FUNCTION_BLOCK P_Call (* Calls one atomic skill: latches P1..P4 on EI, continues on DONE (EO) or FAILED (ERR); ignores completions it did not request *)
  (* Standard: 61499-2 *)
  (* Version 2.0, 2026-09-27, Project contributors, Filling cell reference model *)
  PACKAGE fillingcell;
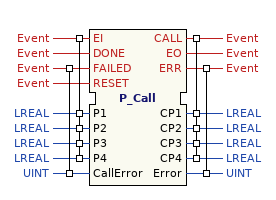
  EVENT_INPUT
    EI WITH P1, P2, P3, P4;
    DONE;
    FAILED WITH CallError;
    RESET;
  END_EVENT
  EVENT_OUTPUT
    CALL WITH CP1, CP2, CP3, CP4;
    EO;
    ERR WITH Error;
  END_EVENT
  VAR_INPUT
    P1 : LREAL;
    P2 : LREAL;
    P3 : LREAL;
    P4 : LREAL;
    CallError : UINT;
  END_VAR
  VAR_OUTPUT
    CP1 : LREAL;
    CP2 : LREAL;
    CP3 : LREAL;
    CP4 : LREAL;
    Error : UINT;
  END_VAR
  VAR
    Busy : BOOL;
  END_VAR
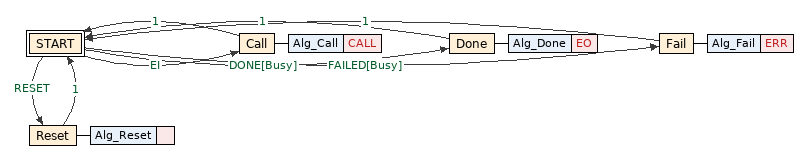
  EC_STATES
    START;
    Call : Alg_Call -> CALL;
    Done : Alg_Done -> EO;
    Fail : Alg_Fail -> ERR;
    Reset : Alg_Reset;
  END_STATES
  EC_TRANSITIONS
    START TO Call := EI;
    START TO Done := DONE[Busy];
    START TO Fail := FAILED[Busy];
    START TO Reset := RESET;
    Call TO START := 1;
    Done TO START := 1;
    Fail TO START := 1;
    Reset TO START := 1;
  END_TRANSITIONS
  ALGORITHM Alg_Call IN ST:
CP1 := P1;
CP2 := P2;
CP3 := P3;
CP4 := P4;
Busy := TRUE;
Error := 0;
  END_ALGORITHM
  ALGORITHM Alg_Done IN ST:
Busy := FALSE;
  END_ALGORITHM
  ALGORITHM Alg_Fail IN ST:
Busy := FALSE;
Error := CallError;
  END_ALGORITHM
  ALGORITHM Alg_Reset IN ST:
Busy := FALSE;
  END_ALGORITHM
END_FUNCTION_BLOCK
